// TwinCAT 3 PLC project ConveyorsLinking
// ProgramVersion: 3.1.4023.0
// libraries:
//   Tc2_Standard, * (Beckhoff Automation GmbH)
//   Tc2_System, * (Beckhoff Automation GmbH)
//   Tc3_Module, * (Beckhoff Automation GmbH)
// project tree:
//   DUTs/ ConveyorLSC.TcPOU (not stored), ConveyorMode.TcDUT (not stored), ConveyorSC.TcPOU (not stored)
//   / PlcTask.TcTTO
//   POUs/ InRange.TcPOU (not stored), MAIN.TcPOU
// real-time tasks:
//   TASK PlcTask: cycle T#10ms, priority 20, ADS port 350
//   TASK PlcTask1: cycle T#10ms, priority 21, ADS port 351
//   TASK PlcTask2: cycle T#10ms, priority 22, ADS port 352
//   TASK PlcTask3: cycle T#10ms, priority 23, ADS port 353

CONFIGURATION ConveyorsLinking
    RESOURCE PLC ON TwinCAT3
        TASK PlcTask(INTERVAL := T#10ms, PRIORITY := 20);
        PROGRAM MAIN WITH PlcTask : MAIN;
    END_RESOURCE
END_CONFIGURATION

// ---- POUs/MAIN.TcPOU
PROGRAM MAIN
VAR
	sc1 : ConveyorSC;
	sc2 : ConveyorSC;
	sc3 : ConveyorSC;
	sc4 : ConveyorSC;
	lsc5 : ConveyorLSC;
	lsc6 : ConveyorLSC;
	lsc7 : ConveyorLSC;
	lsc8 : ConveyorLSC;
	
END_VAR
VAR
	cellConveyors : ARRAY[1..8] OF POINTER TO ConveyorSC;
	
END_VAR
(*
in this module, conveyors are implemented as a linked list
each conveyor's mode is determined by the actual mode (not requested mode) of its adjacent conveyors
*)

//double click on these for online write
(*
conveyor linking algorithm:
	-find a chain where all conveyors are occupied
	-find highest priority request between the chain
	-set the actual mode all conveyors in the chain to that highest priority request
*)

call();

sc1.trueMode;
sc2.trueMode;
sc3.trueMode;
sc4.trueMode;
lsc5.trueMode;
lsc6.trueMode;
lsc7.trueMode;
lsc8.trueMode;

sc1.requestedMode;
sc2.requestedMode;
sc3.requestedMode;
sc4.requestedMode;
lsc5.requestedMode;
lsc6.requestedMode;
lsc7.requestedMode;
lsc8.requestedMode;

slowLink();
//fastLink();





call();

METHOD call : BOOL
VAR_INPUT
END_VAR
VAR
	i : INT;
END_VAR
cellConveyors[1] := ADR(sc1);
cellConveyors[2] := ADR(sc2);
cellConveyors[3] := ADR(sc3);
cellConveyors[4] := ADR(sc4);
cellConveyors[5] := ADR(lsc5);
cellConveyors[6] := ADR(lsc6);
cellConveyors[7] := ADR(lsc7);
cellConveyors[8] := ADR(lsc8);

FOR i:=1 TO 8-1 BY 1 DO
	
	cellConveyors[i]^.join(cellConveyors[i+1]);
	
END_FOR


sc1(error=> , position=> , velocity=> );
sc2(error=> , position=> , velocity=> );
sc3(error=> , position=> , velocity=> );
sc4(error=> , position=> , velocity=> );

lsc5(
	error=> , 
	position=> , 
	velocity=> , 
	lifterError=> , 
	extended=> , 
	retracted=> );
	
lsc6(
	error=> , 
	position=> , 
	velocity=> , 
	lifterError=> , 
	extended=> , 
	retracted=> );
	
lsc7(
	error=> , 
	position=> , 
	velocity=> , 
	lifterError=> , 
	extended=> , 
	retracted=> );
	
lsc8(
	error=> , 
	position=> , 
	velocity=> , 
	lifterError=> , 
	extended=> , 
	retracted=> );
END_METHOD

METHOD fastLink : BOOL
VAR
	i : INT;
	j : INT;
	
	linkStart : INT := -1;
	linkEnd : INT := -1;
	
	priorityInLink : ConveyorMode;
END_VAR
VAR
	numLinks : INT;
	
	startLinks : ARRAY[0..numCellConveyors-1] OF INT := [numCellConveyors(-1)];
	endLinks : ARRAY[0..numCellConveyors-1] OF INT := [numCellConveyors(-1)];
	chainPriority : ARRAY[0..numCellConveyors] OF ConveyorMode := [numCellConveyors(ConveyorMode.IDLE)];
	
	iLinkSetter : INT;
END_VAR
VAR CONSTANT
	numCellConveyors : INT := 8;
END_VAR
FOR i:=1 TO numCellConveyors BY 1 DO
	
	IF cellConveyors[i]^.IsOccupied THEN
		
		IF linkStart = -1 THEN
			startLinks[numLinks] := i;
		END_IF
		
		chainPriority[numLinks] := MAX(priorityInLink, cellConveyors[i]^.requestedMode);
		endLinks[numLinks] := i;
		
	ELSIF linkStart <> -1 AND linkEnd <> -1 THEN //set the link end index and increment number of links
		
		endLinks[numLinks] := i-1;
		numLinks := numLinks + 1;
		
	END_IF
	
END_FOR

//final link
IF startLinks[numLinks] > -1 AND endLinks[numLinks] > -1 THEN
	endLinks[numLinks] := i;
	numLinks := numLinks + 1;
END_IF

//set the true modes to all conveyors
FOR i:=1 TO numCellConveyors BY 1 DO
	
	IF iLinkSetter < numLinks AND InRange(v1:= startLinks[iLinkSetter], v2:= endLinks[iLinkSetter], value:= i, inclusive:= TRUE) THEN
		
		cellConveyors[i]^.setMode(mode:= chainPriority[iLinkSetter]);
		IF i = endLinks[iLinkSetter] THEN
			iLinkSetter := iLinkSetter + 1;
		END_IF
		
	END_IF
	
END_FOR
END_METHOD

METHOD slowLink : BOOL
VAR_INPUT
END_VAR
VAR
	i : INT;
	j : INT;
	
	linkStart : INT := -1;
	linkEnd : INT := -1;
	chainMode : ConveyorMode;
END_VAR
linkStart := -1;
linkEnd := -1;
chainMode := 0;

FOR i:=1 TO 8 BY 1 DO
	
	IF cellConveyors[i]^.IsOccupied THEN
		IF linkStart = -1 THEN
			linkStart := i;
		END_IF
		
		chainMode := MAX(chainMode, cellConveyors[i]^.requestedMode);
		linkEnd := i;
	
	ELSIF linkStart <> -1 AND linkEnd <> -1 THEN //set all conveyor operations to priorityInLink
		
		FOR j:=linkStart TO linkEnd BY 1 DO
			cellConveyors[j]^.setMode(chainMode);
		END_FOR
		
		linkStart := -1;
		linkEnd := -1;
		
		chainMode := ConveyorMode.IDLE;
		cellConveyors[i]^.setMode(ConveyorMode.IDLE);
		
		CONTINUE;
	END_IF
	
END_FOR

IF linkStart > -1 AND linkEnd > -1 THEN
	FOR j:=linkStart TO linkEnd BY 1 DO
		cellConveyors[j]^.setMode(chainMode);
	END_FOR
END_IF
END_METHOD

END_PROGRAM
